FUNCTION_BLOCK goToAbsPos (* Composite Function Block Type *)
  (* Standard: 61499-2 *)
  (* Version 1.0, 2019-05-27, Promok *)
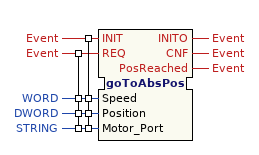
  EVENT_INPUT
    INIT WITH Speed, Motor_Port, Position; (* Initialization Request *)
    REQ WITH Speed, Motor_Port, Position; (* Normal Execution Request *)
  END_EVENT
  EVENT_OUTPUT
    INITO; (* Initialization Confirm *)
    CNF; (* Execution Confirmation *)
    PosReached; (* Position Reached *)
  END_EVENT
  VAR_INPUT
    Speed : WORD; (* Set Motor Speed *)
    Position : DWORD; (* Set target absolute position *)
    Motor_Port : STRING; (* Set motor port *)
  END_VAR
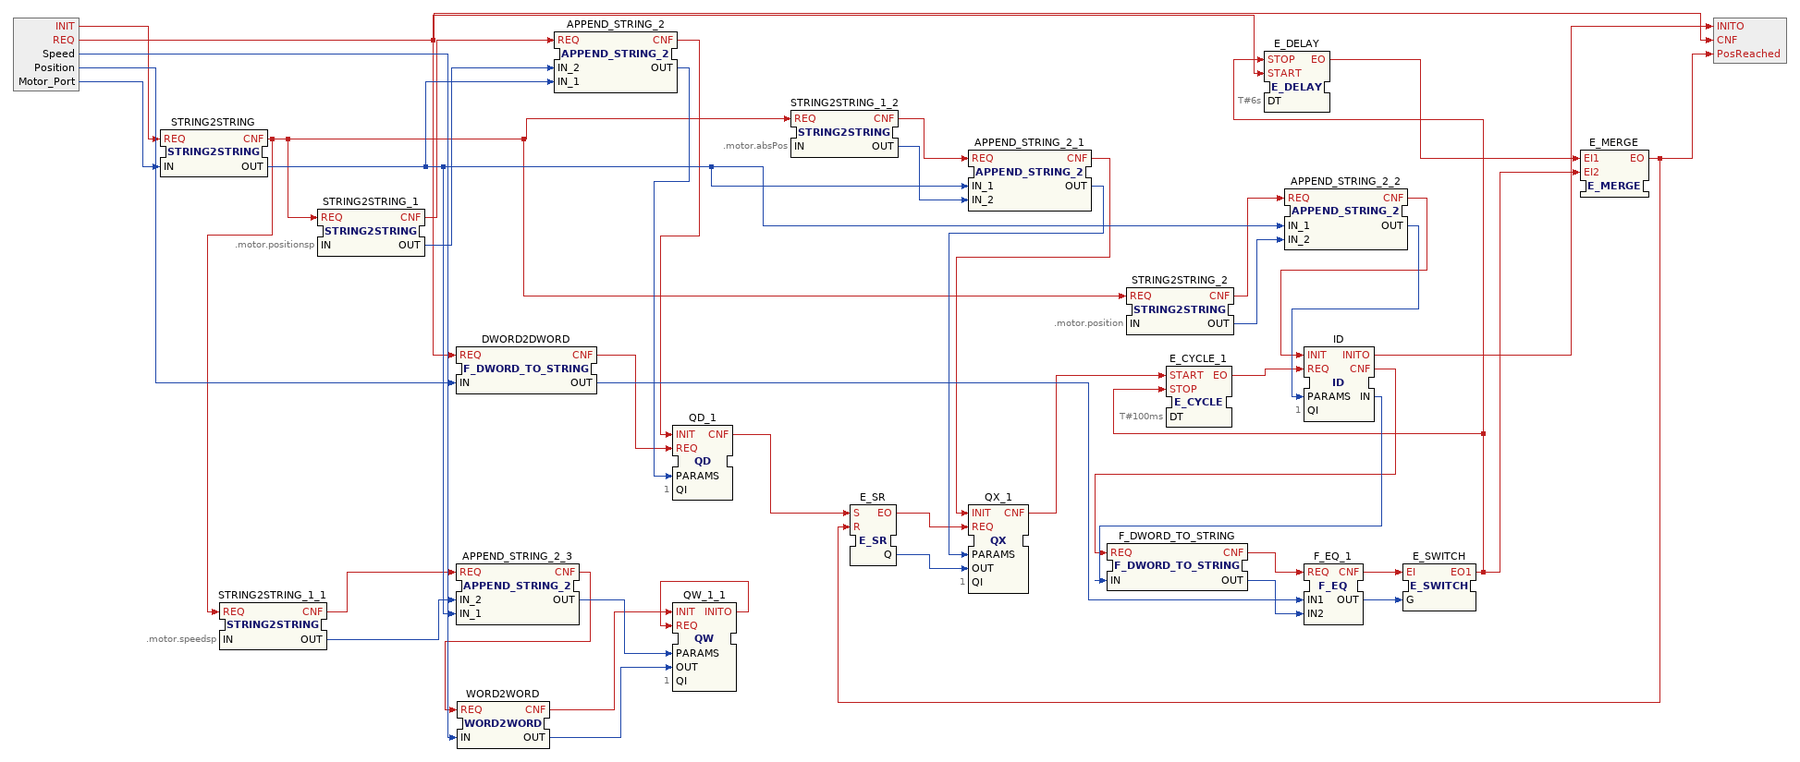
  FBS
    WORD2WORD : WORD2WORD;
    F_EQ_1 : F_EQ;
    ID : ID(QI := 1);
    APPEND_STRING_2_1 : APPEND_STRING_2;
    QX_1 : QX(QI := 1);
    STRING2STRING : STRING2STRING;
    APPEND_STRING_2 : APPEND_STRING_2;
    E_CYCLE_1 : E_CYCLE(DT := T#100ms);
    QD_1 : QD(QI := 1);
    STRING2STRING_1_1 : STRING2STRING(IN := .motor.speedsp);
    APPEND_STRING_2_3 : APPEND_STRING_2;
    E_SWITCH : E_SWITCH;
    STRING2STRING_1_2 : STRING2STRING(IN := .motor.absPos);
    STRING2STRING_1 : STRING2STRING(IN := .motor.positionsp);
    QW_1_1 : QW(QI := 1);
    APPEND_STRING_2_2 : APPEND_STRING_2;
    STRING2STRING_2 : STRING2STRING(IN := .motor.position);
    E_DELAY : E_DELAY(DT := T#6s);
    E_SR : E_SR;
    E_MERGE : E_MERGE;
    DWORD2DWORD : F_DWORD_TO_STRING;
    F_DWORD_TO_STRING : F_DWORD_TO_STRING;
  END_FBS
  EVENT_CONNECTIONS
    APPEND_STRING_2_2.CNF TO ID.INIT;
    APPEND_STRING_2_3.CNF TO WORD2WORD.REQ;
    E_CYCLE_1.EO TO ID.REQ;
    STRING2STRING.CNF TO STRING2STRING_2.REQ;
    STRING2STRING_1.CNF TO APPEND_STRING_2.REQ;
    STRING2STRING_2.CNF TO APPEND_STRING_2_2.REQ;
    STRING2STRING.CNF TO STRING2STRING_1.REQ;
    QX_1.CNF TO E_CYCLE_1.START;
    E_SWITCH.EO1 TO E_CYCLE_1.STOP;
    APPEND_STRING_2.CNF TO QD_1.INIT;
    STRING2STRING.CNF TO STRING2STRING_1_2.REQ;
    WORD2WORD.CNF TO QW_1_1.INIT;
    STRING2STRING_1_1.CNF TO APPEND_STRING_2_3.REQ;
    F_EQ_1.CNF TO E_SWITCH.EI;
    STRING2STRING.CNF TO STRING2STRING_1_1.REQ;
    QW_1_1.INITO TO QW_1_1.REQ;
    APPEND_STRING_2_1.CNF TO QX_1.INIT;
    STRING2STRING_1_2.CNF TO APPEND_STRING_2_1.REQ;
    REQ TO CNF;
    ID.INITO TO INITO;
    E_SWITCH.EO1 TO E_DELAY.STOP;
    REQ TO E_DELAY.START;
    QD_1.CNF TO E_SR.S;
    E_SR.EO TO QX_1.REQ;
    E_DELAY.EO TO E_MERGE.EI1;
    E_SWITCH.EO1 TO E_MERGE.EI2;
    E_MERGE.EO TO PosReached;
    E_MERGE.EO TO E_SR.R;
    INIT TO STRING2STRING.REQ;
    REQ TO DWORD2DWORD.REQ;
    DWORD2DWORD.CNF TO QD_1.REQ;
    ID.CNF TO F_DWORD_TO_STRING.REQ;
    F_DWORD_TO_STRING.CNF TO F_EQ_1.REQ;
  END_CONNECTIONS
  DATA_CONNECTIONS
    APPEND_STRING_2_3.OUT TO QW_1_1.PARAMS;
    STRING2STRING_1_1.OUT TO APPEND_STRING_2_3.IN_2;
    APPEND_STRING_2_2.OUT TO ID.PARAMS;
    APPEND_STRING_2.OUT TO QD_1.PARAMS;
    STRING2STRING.OUT TO APPEND_STRING_2_1.IN_1;
    F_EQ_1.OUT TO E_SWITCH.G;
    STRING2STRING_1.OUT TO APPEND_STRING_2.IN_2;
    STRING2STRING.OUT TO APPEND_STRING_2.IN_1;
    WORD2WORD.OUT TO QW_1_1.OUT;
    APPEND_STRING_2_1.OUT TO QX_1.PARAMS;
    STRING2STRING.OUT TO APPEND_STRING_2_2.IN_1;
    STRING2STRING_2.OUT TO APPEND_STRING_2_2.IN_2;
    STRING2STRING_1_2.OUT TO APPEND_STRING_2_1.IN_2;
    STRING2STRING.OUT TO APPEND_STRING_2_3.IN_1;
    Motor_Port TO STRING2STRING.IN;
    Speed TO WORD2WORD.IN;
    E_SR.Q TO QX_1.OUT;
    Position TO DWORD2DWORD.IN;
    DWORD2DWORD.OUT TO F_EQ_1.IN1;
    ID.IN TO F_DWORD_TO_STRING.IN;
    F_DWORD_TO_STRING.OUT TO F_EQ_1.IN2;
  END_CONNECTIONS
END_FUNCTION_BLOCK
